TYPE ST_AmbientState :
STRUCT
	fOutsideTemperature : REAL;
	fHallTemperature : REAL;
	bRain : BOOL;
END_STRUCT
END_TYPE

(* stored: Version 1.1.0.1, ProductVersion 3.1.4024.10
   DUT ST_AmbientState: Id {18024053-1db6-499b-af8a-99fd20169e28} *)
